PROGRAM Belt_and_Gripper
VAR
	STATUS : BOOL;
END_VAR

IF STATUS = TRUE THEN
	;
END_IF

END_PROGRAM

(* stored: Version 1.1.0.1, ProductVersion 3.1.4024.15
   POU Belt_and_Gripper: Id {9ead365b-d204-4444-b5a5-da437d7e747f}, SpecialFunc None *)
